FUNCTION_BLOCK ProcessDataManager EXTENDS TcoData.TcoDataExchange
VAR
    _data : ProcessData := (Parent := THIS^);
END_VAR

SUPER^();

PROPERTY Data : REFERENCE TO ProcessData
GET
Data REF= _data;
END_GET
END_PROPERTY

END_FUNCTION_BLOCK

(* stored: Version 1.1.0.1, ProductVersion 3.1.4024.9
   POU ProcessDataManager: Id {2c1ab05b-163f-4701-a4e6-85eef79998c1}, SpecialFunc None
   Property Data: Id {40710a68-4852-4e7f-af06-13ca5d713a1b}
   Get Get: Id {7ffb2cbf-81a9-4de7-9388-60f1b13fbd72} *)
